// TIA Portal V15.1 export
// export: Created 2022-12-20T09:13:22.053784Z, ExportSetting None, DisplayName Totally Integrated Automation Portal, DisplayVersion V15.1 Update 1, DisplayName TIA Portal Openness, DisplayVersion V15.1, DisplayName SINAMICS Startdrive Advanced, DisplayVersion V15.1, DisplayName G130, G150, S120, S150, SINAMICS MV, S210, DisplayVersion V15.1, DisplayName G110M, G120, G120C, G120D, G120P, DisplayVersion V15.1, DisplayName STEP 7 Professional, DisplayVersion V15.1 Update 1, DisplayName STEP 7 Safety, DisplayVersion V15.1, DisplayName WinCC Professional, DisplayVersion V15.1 Update 1, DisplayName SIMATIC Visualization Architect, DisplayVersion V15.1
FUNCTION_BLOCK "SA01_EM11_++xxx+xxxx_FB"   // FB1110, FBD
TITLE = SA01_EM11_++xxx+xxxx_FB
{ S7_Optimized_Access := 'FALSE' }
// The block is used to control EM11 Fixture xxx+xxxx and all its associated CMs
// stored: AutoNumber false, SetENOAutomatically False
   VAR
      Mode : "Mode_EM_FB";   // Mode
      "xxx-xxxx" : "Type_Lookup_FB";   // xxxxx
   END_VAR
BEGIN

REGION Network 1: ***Mode***
END_REGION

REGION Network 2: Mode settings
   // Setting holding to held
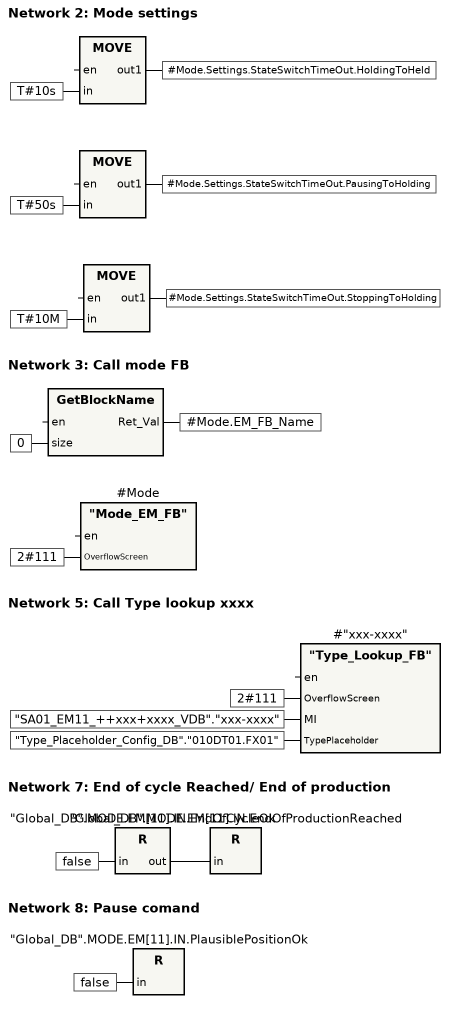
   #Mode.Settings.StateSwitchTimeOut.HoldingToHeld := T#10s;
   #Mode.Settings.StateSwitchTimeOut.PausingToHolding := T#50s;
   #Mode.Settings.StateSwitchTimeOut.StoppingToHolding := T#10M;
END_REGION

REGION Network 3: Call mode FB
   // Depending on the inputs preconditions, commands, alarms, HMI and input from Safety Area (SA) Determine the current function, mode of operandi, and state.
   #Mode.EM_FB_Name := GetBlockName(size := 0);
   #Mode(OverflowScreen := 2#111);   // "Mode_EM_FB"
END_REGION

REGION Network 4: ***TYPE***
END_REGION

REGION Network 5: Call Type lookup xxxx
   // Type xxxxx
   #"xxx-xxxx"(OverflowScreen := 2#111,   // "Type_Lookup_FB"
               MI := "SA01_EM11_++xxx+xxxx_VDB"."xxx-xxxx",
               TypePlaceholder := "Type_Placeholder_Config_DB"."010DT01.FX01");
END_REGION

REGION Network 6: **Process status**
END_REGION

REGION Network 7: End of cycle Reached/ End of production
   // no phase active
   IF false THEN
       "Global_DB".MODE.EM[11].IN.EndOfCycleOk := FALSE;
       "Global_DB".MODE.EM[11].IN.EndOfProductionReached := FALSE;
   END_IF;
END_REGION

REGION Network 8: Pause comand
   // Pause comand
   IF false THEN "Global_DB".MODE.EM[11].IN.PlausiblePositionOk := FALSE; END_IF;
END_REGION
END_FUNCTION_BLOCK
